{attribute 'qualified_only'}
{attribute 'strict'}
TYPE EnumState :
(
	init,
	drive1,
	drive2,
	reset
);
END_TYPE

(* stored: Version 1.1.0.1, ProductVersion 3.1.4022.3
   DUT EnumState: Id {31591028-10a2-478a-84f1-4f97ed464496} *)
